{region '#Template'}
	{attribute 'Version' := '1.0.1.0'}
	{attribute 'Tags' := '"LCID": "1031", "Text": "AC, Aggregates, pre-heater, Return temperature control"'}
	{attribute 'Tags' := '"LCID": "1033", "Text": "AC, Aggregates, pre-heater, Return temperature control"'}
	{attribute 'Description' := '"LCID": "1031", "Text": "Vorerhitzer Rücklauf Temperatur Regelung"'}
	{attribute 'Description' := '"LCID": "1033", "Text": "Pre-Heater return temperature control"'}
{endregion}
FUNCTION_BLOCK FB_BA_AC_TRtCtrl EXTENDS FB_BA_View
VAR_INPUT
	bActivatePreRinse		: BOOL;
	fTRt					: REAL;
	bTWthLowLimit			: BOOL;
	fTWth					: REAL;
	bSuACtrlSeqActive		: BOOL;
	bMixADmpAvail			: BOOL;
END_VAR
VAR_OUTPUT
	fY						: REAL;
	bPreRinseActive			: BOOL;
	bPreRinseDstb			: BOOL;
END_VAR
VAR_INPUT CONSTANT
	SpTRtW					: FB_BA_AV_Op;
	PreRinseDelay			: FB_BA_DlyOn;												 
	PreRinseDst				: FB_BA_BV;													   
	PreRinseSp				: FB_BA_Scale_02;																		
	Ctrl					: FB_BA_LoopSeq;	
END_VAR
VAR
	bPreRinseReady			: BOOL;
	rtrigActivatePreRinse	: R_TRIG;
	rsPreRinse				: RS;
	rsPreRinseActive		: RS;
	rsSelSp					: RS;
	PreRinseHys				: FB_BA_Swi2P;
END_VAR

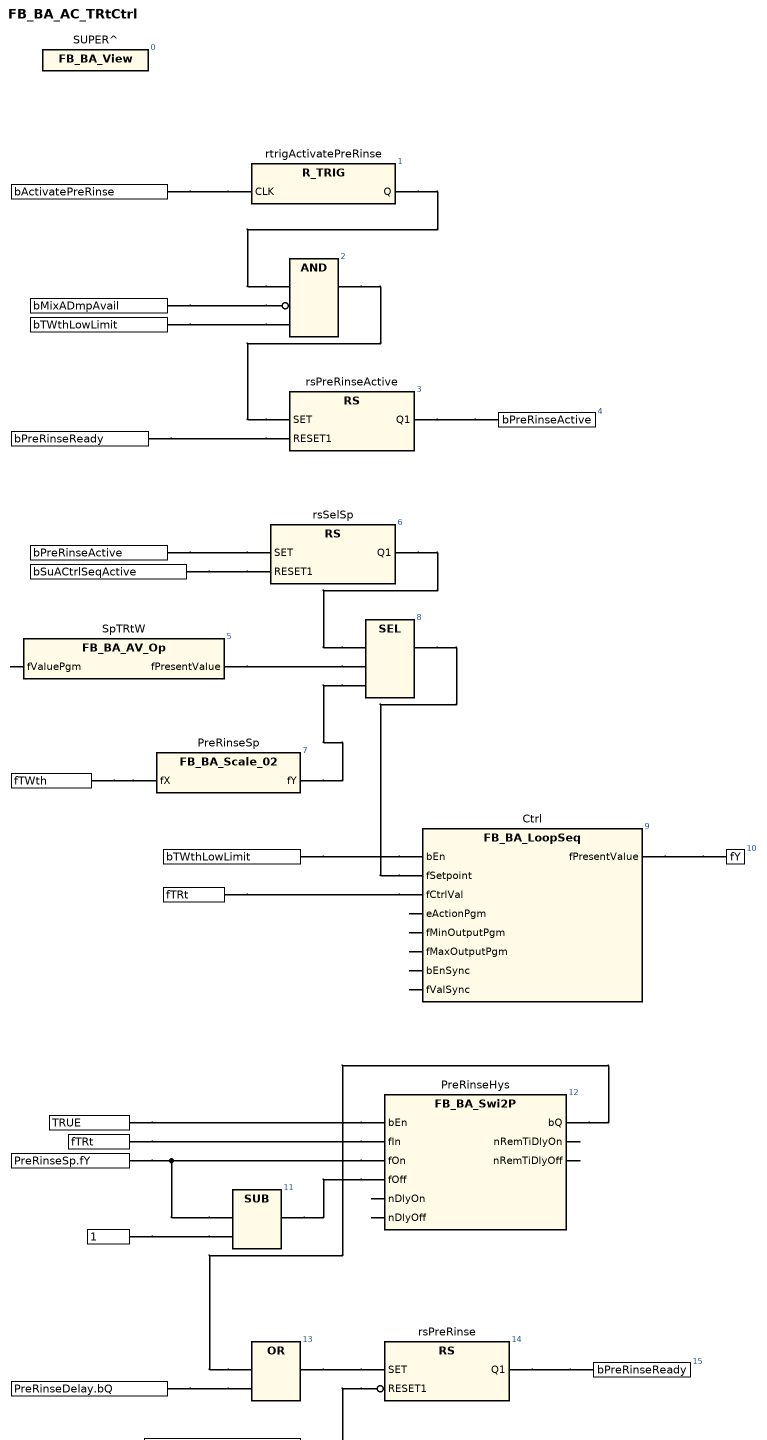
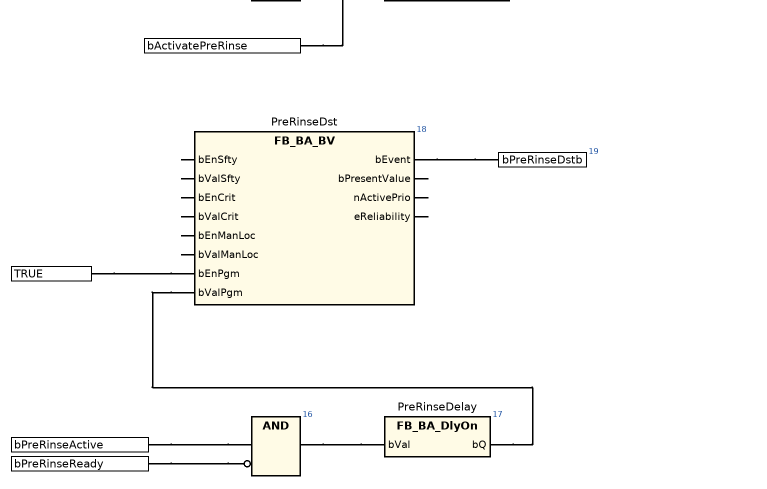
SUPER^(); // FB_BA_View
rtrigActivatePreRinse(CLK := bActivatePreRinse); // R_TRIG
rsPreRinseActive(SET := rtrigActivatePreRinse.Q AND NOT bMixADmpAvail AND bTWthLowLimit, RESET1 := bPreRinseReady); // RS
bPreRinseActive := rsPreRinseActive.Q1;
SpTRtW(); // FB_BA_AV_Op
rsSelSp(SET := bPreRinseActive, RESET1 := bSuACtrlSeqActive); // RS
PreRinseSp(fX := fTWth); // FB_BA_Scale_02
Ctrl(
    bEn := bTWthLowLimit,
    fSetpoint := SEL(rsSelSp.Q1, SpTRtW.fPresentValue, PreRinseSp.fY),
    fCtrlVal := fTRt); // FB_BA_LoopSeq
fY := Ctrl.fPresentValue;
PreRinseHys(bEn := TRUE, fIn := fTRt, fOn := PreRinseSp.fY, fOff := PreRinseSp.fY - 1); // FB_BA_Swi2P
rsPreRinse(SET := PreRinseHys.bQ OR PreRinseDelay.bQ, RESET1 := NOT bActivatePreRinse); // RS
bPreRinseReady := rsPreRinse.Q1;
PreRinseDelay(bVal := bPreRinseActive AND NOT bPreRinseReady); // FB_BA_DlyOn
// parameter PreRinseDst.bValManualRm := TRUE
PreRinseDst(bEnPgm := TRUE, bValPgm := PreRinseDelay.bQ); // FB_BA_BV
bPreRinseDstb := PreRinseDst.bEvent;

METHOD FB_init : BOOL
VAR_INPUT
	bInitRetains : BOOL; // if TRUE, the retain variables are initialized (warm start / cold start)
	bInCopyCode : BOOL;  // if TRUE, the instance afterwards gets moved into the copy code (online change)
END_VAR
SpTRtW.iParent								:= THIS^;
SpTRtW.iLabel								:= LblCmpAC.PreHtr_TRtCtrl_SpTRtW;
SpTRtW.sObjectName							:= '{Idx=01}';	
SpTRtW.eUnit 								:= E_BA_Unit.eTemperature_DegreesCelsius;								 								
SpTRtW.fValueRm								:= 5.0;

PreRinseDelay.iParent						:= THIS^;	
PreRinseDelay.iLabel						:= LblCmpAC.PreHtr_TRtCtrl_PreRinseDelay;
PreRinseDelay.sObjectName					:= '{Idx=01}';				
PreRinseDelay.eDPADMode						:= E_BA_DPADMode.eIncludeDescription;
PreRinseDelay.TiDly.iLabel					:= LblCmpAC.PreHtr_TRtCtrl_PreRinseDelay_TiDly;
PreRinseDelay.TiDly.fValueRm				:= 900;	

PreRinseDst.iParent							:= THIS^;
PreRinseDst.iLabel							:= LblCmpAC.PreHtr_TRtCtrl_PreRinseDst;			
PreRinseDst.sObjectName						:= '{Idx=01}';	
PreRinseDst.bEnOutOfService					:= FALSE;
PreRinseDst.sActiveText 					:= txtEvent_Triggered;
PreRinseDst.sInactiveText 					:= txtEvent_Normal;
PreRinseDst.nStateChangeCount				:= 0;
PreRinseDst.nActiveTimeElapsed				:= 0;
PreRinseDst.nMinimumOnTime					:= 0;
PreRinseDst.nMinimumOffTime					:= 0;
PreRinseDst.bEnManualRm						:= FALSE;	//	Priority  8	
PreRinseDst.bValManualRm					:= FALSE;	//	Priority  8
PreRinseDst.bDefaultValue					:= FALSE;
PreRinseDst.nEventClassID					:= EventClasses.AlarmTechnicalExtended;
PreRinseDst.stTimeDelay.nToNormal			:= BA2_Param.nDefTimeDelay_ToNormal;
PreRinseDst.stTimeDelay.nToAbnormal			:= BA2_Param.nDefTimeDelay_ToAbnormal;
PreRinseDst.bAlarmValue						:= TRUE;
PreRinseDst.bAcknowledgeRm					:= FALSE;		
PreRinseDst.aEventTransitionText[1]			:= txtEvent_Triggered;
PreRinseDst.aEventTransitionText[2]			:= txtEvent_Error;
PreRinseDst.aEventTransitionText[3]			:= txtEvent_Normal;
PreRinseDst.bEventDetectionEnable			:= TRUE;
PreRinseDst.eEnPlantLock					:= E_BA_LockPriority.eNoLock;	

PreRinseSp.iParent							:= THIS^;
PreRinseSp.iLabel							:= LblCmpAC.PreHtr_TRtCtrl_PreRinseSp;			
PreRinseSp.sObjectName						:= '{Idx=02}';
PreRinseSp.eDPADMode						:= E_BA_DPADMode.eIncludeDescription;
PreRinseSp.X1.fValueRm						:= 10.0;
PreRinseSp.X2.fValueRm						:= 0.0;
PreRinseSp.Y1.fValueRm						:= 25.0;
PreRinseSp.Y2.fValueRm						:= 45.0;
PreRinseSp.YMin.fValueRm					:= 20.0;
PreRinseSp.YMax.fValueRm					:= 60.0;

Ctrl.iParent								:= THIS^;
Ctrl.iLabel									:= LblCmpAC.PreHtr_TRtCtrl_Ctrl; 
Ctrl.sObjectName							:= '{Idx=01}';
Ctrl.eOpMode								:= BA2_Param.nLoop_DefOpMode;								 	 										 
Ctrl.eOutputUnit							:= E_BA_Unit.eOther_Percent;
Ctrl.eActionRm								:= E_BA_Action.eReverse;
Ctrl.fProportionalConstant					:= 3;
Ctrl.fIntegralConstant						:= 180;
Ctrl.fDerivativeConstant					:= 0;
Ctrl.fMaxOutputRm 							:= 100;
Ctrl.fMinOutputRm							:= 0;
Ctrl.fCOVIncrement							:= 0;
Ctrl.nDampConstant							:= 0;
Ctrl.fNeutralZone							:= 0;
END_METHOD

END_FUNCTION_BLOCK

(* stored: Version 1.1.0.1, ProductVersion 3.1.4024.9
   POU FB_BA_AC_TRtCtrl: Id {00000000-0000-0000-0000-000000000000}, SpecialFunc None
   Method FB_init: Id {2786c226-9c64-4c1e-868c-4b2ad6341ea5} *)
